TEXTLIST EL2809_M_2
  1 = 'Unwinding L Brake' | chinese: '放卷L_刹车' | Chinese: '放卷L_刹车'
  2 = 'Un_L Clutch Out' | chinese: '放卷L_离合器out' | Chinese: '放卷L_离合器out'
  3 = 'Un_L Clutch RST' | chinese: '放卷L_离合器rst' | Chinese: '放卷L_离合器rst'
  4 = 'Un_R Brake' | chinese: '放卷R_刹车' | Chinese: '放卷R_刹车'
  5 = 'Un_R Clutch Out' | chinese: '放卷R_离合器out' | Chinese: '放卷R_离合器out'
  6 = 'Un_R Clutch RST' | chinese: '放卷R_离合器rst' | Chinese: '放卷R_离合器rst'
  7 = 'Re_L Clutch Out' | chinese: '收卷L_离合器out' | Chinese: '收卷L_离合器out'
  8 = 'Re_L Clutch RST' | chinese: '收卷L_离合器rst' | Chinese: '收卷L_离合器rst'
  9 = 'Re_R Clutch Out' | chinese: '收卷R_离合器out' | Chinese: '收卷R_离合器out'
  10 = 'Re_R Clutch RST' | chinese: '收卷R_离合器rst' | Chinese: '收卷R_离合器rst'
  11 = 'S1 Drive enabled' | chinese: '导向压轮电机使能' | Chinese: '导向压轮电机使能'
  12 = 'S1 Forward/Reverse' | chinese: '导向压轮电机正/反转' | Chinese: '导向压轮电机正/反转'
  13 = 'S1_Break' | chinese: '导向压轮电机刹车' | Chinese: '导向压轮电机刹车'
  14 = ''
  15 = ''
  16 = ''
   = ''
END_TEXTLIST

(* stored: Version 1.1.0.1, ProductVersion 3.1.4024.11
   TextList EL2809_M_2: Id {98433cd8-49a2-44d4-bbb3-34237b80c705} *)
